// TIA Portal V17 export
// export: Created 2022-04-06T07:28:40.5956823Z, ExportSetting WithDefaults, DisplayName Totally Integrated Automation Portal, DisplayVersion V17, DisplayName TIA Portal Openness, DisplayVersion V17, DisplayName TIA Portal Version Control Interface, DisplayVersion V17, DisplayName TIA Portal Test Suite Advanced, DisplayVersion V17, DisplayName SINAMICS Startdrive Advanced, DisplayVersion V17, DisplayName SINAMICS Startdrive G130, G150, S120, S150, SINAMICS MV, S210, DisplayVersion V17, DisplayName SINAMICS Startdrive G110M, G120, G120C, G120D, G120P, G115D, DisplayVersion V17, DisplayName STEP 7 Professional, DisplayVersion V17, DisplayName STEP 7 Safety, DisplayVersion V17, DisplayName WinCC Advanced / Unified PC, DisplayVersion V17
TYPE "LDrvSafe_typeSinaTlg901Status"
TITLE = LDrvSafe_typeSinaTlg901Status
// Failsafe user-defined data type for PROFIsafe telegram 901 to get status information of Safety Integrated Functions of SINAMICS
// stored: IsFailsafeCompliant true
   STRUCT
      STOactive { ExternalWritable := 'False'} : Bool;   // Safety Function Safe Torque Off active
      SS1active { ExternalWritable := 'False'} : Bool;   // Safety Function Safe Stop 1 active
      SS2active { ExternalWritable := 'False'} : Bool;   // Safety Function Safe Stop 2 active
      SOSactive { ExternalWritable := 'False'} : Bool;   // Safety Function Safe Operating Stop active
      SLSactive { ExternalWritable := 'False'} : Bool;   // Safety Function Safely-limited Speed active
      reserved1 { ExternalWritable := 'False'} : Bool;   // Reserve bit 1
      SLPactive { ExternalWritable := 'False'} : Bool;   // Safety Function Safely-limited Position active
      internalEvent { ExternalWritable := 'False'} : Bool;   // Internal Event occured (Safety error in SINAMICS)
      SLAactive { ExternalWritable := 'False'} : Bool;   // Safety Function Safely-limited Acceleration active
      SLSbit0Active { ExternalWritable := 'False'} : Bool;   // One of the the four SLS limits is active; operates together with bit 1
      SLSbit1Active { ExternalWritable := 'False'} : Bool;   // One of the the four SLS limits is active; operates together with bit 0
      reserved3 { ExternalWritable := 'False'} : Bool;   // Reserve bit 3
      SDIpositiveActive { ExternalWritable := 'False'} : Bool;   // Safety Function Safe Direction (positive direction) active
      SDInegativeActive { ExternalWritable := 'False'} : Bool;   // Safety Function Safe Direction (negative direction) active
      reserved4 { ExternalWritable := 'False'} : Bool;   // Reserve bit 4
      SSMactive { ExternalWritable := 'False'} : Bool;   // Safety Function Safe Speed Monitor; signals, if safe speed is below paramterizable speed limit
      reserved5 { ExternalWritable := 'False'} : Bool;   // Reserve bit 5
      reserved6 { ExternalWritable := 'False'} : Bool;   // Reserve bit 6
      reserved7 { ExternalWritable := 'False'} : Bool;   // Reserve bit 7
      SLPrangeActive { ExternalWritable := 'False'} : Bool;   // SLP position range 1 or 2 is active
      reserved8 { ExternalWritable := 'False'} : Bool;   // Reserve bit 8
      reserved9 { ExternalWritable := 'False'} : Bool;   // Reserve bit 9
      safePositionValid { ExternalWritable := 'False'} : Bool;   // Safe Position is valid
      safelyReferenced { ExternalWritable := 'False'} : Bool;   // Drive is safely referenced
      statusFDI0 { ExternalWritable := 'False'} : Bool;   // Status of Failsafe Digital Input 0
      statusFDI1 { ExternalWritable := 'False'} : Bool;   // Status of Failsafe Digital Input 1
      statusFDI2 { ExternalWritable := 'False'} : Bool;   // Status of Failsafe Digital Input 2
      reserved10 { ExternalWritable := 'False'} : Bool;   // Reserve bit 10
      SS2Eactive { ExternalWritable := 'False'} : Bool;   // Safety Function SS2E active
      SOSselected { ExternalWritable := 'False'} : Bool;   // Safety Function Safe Operating Stop selected (not active yet)
      SLPupperLimitMaintained { ExternalWritable := 'False'} : Bool;   // SLP: upper limit maintained
      SLPlowerLimitMaintained { ExternalWritable := 'False'} : Bool;   // SLP: lower limit maintained
      variableSLSvalue { ExternalWritable := 'False'} : Int;   // Actual SLS value for SLS limit 1
      cycleCounter { ExternalWritable := 'False'} : Int;   // Counter for the Safety cycle
      safePosition { ExternalWritable := 'False'} : Int;   // Current actual position value
   END_STRUCT;
END_TYPE
